// TIA Portal project "s7_1200_1214DCDCDC_loadcell_advanced" (V17)

(* hardware
DEVICE "S7-1200 station_1"  S7-1200 Station
   slot 0: "Rack_0"  S7-1200 Rack  Rack  V1.0
   slot 1: "PLC_1"  CPU 1214C DC/DC/DC  6ES7 214-1AG40-0XB0  V4.2
*)

// ===== PLC "PLC_1"  CPU 1214C DC/DC/DC =====

VAR_GLOBAL   // PLC tag table "Default tag table"
   "Start" AT %I0.2 : Bool;
   "Stop" AT %I0.3 : Bool;
   "Sensor_loadcell_in" AT %IW64 : UInt;
   "Sensor_Loadcell" AT %I0.4 : Bool;
   "Sensor_Classification" AT %I0.5 : Bool;
   "Cylinder_Push" AT %Q0.1 : Bool;
   "Cylinder_GoBack" AT %Q0.2 : Bool;
   "VEL" AT %MW160 : Int;
   "Tag_1" AT %M0.0 : Bool;
   "Tag_2" AT %M0.1 : Bool;
   "Tag_3" AT %M0.2 : Bool;
   "Tag_4" AT %M0.3 : Bool;
   "Tag_5" AT %M0.4 : Bool;
   "Sensor_Mass_Dectect" AT %I0.6 : Bool;
   "Tag_6" AT %M0.5 : Bool;
   "Tag_7" AT %M0.6 : Bool;
   "Tag_8" AT %MD20 : Real;
   "Tag_9" AT %MD30 : Real;
   "Tag_10" AT %MD40 : Real;
   "Tag_11" AT %MD50 : DInt;
   "Mass" AT %MW10 : Word;
   "System_Byte" AT %MB1 : Byte;
   "FirstScan" AT %M1.0 : Bool;
   "DiagStatusUpdate" AT %M1.1 : Bool;
   "AlwaysTRUE" AT %M1.2 : Bool;
   "AlwaysFALSE" AT %M1.3 : Bool;
   "Clock_Byte" AT %MB2 : Byte;
   "Clock_10Hz" AT %M2.0 : Bool;
   "Clock_5Hz" AT %M2.1 : Bool;
   "Clock_2.5Hz" AT %M2.2 : Bool;
   "Clock_2Hz" AT %M2.3 : Bool;
   "Clock_1.25Hz" AT %M2.4 : Bool;
   "Clock_1Hz" AT %M2.5 : Bool;
   "Clock_0.625Hz" AT %M2.6 : Bool;
   "Clock_0.5Hz" AT %M2.7 : Bool;
   "Tag_12" AT %MW12 : UInt;
   "Tag_13" AT %MW14 : UInt;
   "Counter" AT %MB10 : USInt;
   "Aver_val" AT %MW16 : UInt;
   "Tag_14" AT %MD44 : Real;
   "Tag_29" AT %MD48 : Real;
   "Tag_15" AT %M0.7 : Bool;
   "Tag_16" AT %MW18 : Word;
   "CV" AT %MD52 : Real;
   "Tag_20" AT %MD56 : Real;
   "RL_chan" AT %M3.1 : Bool;
   "RL_le" AT %M3.2 : Bool;
   "Tag_23" AT %M3.3 : Bool;
   "Tag_24" AT %M3.4 : Bool;
   "Tag_25" AT %MD60 : Real;
   "Tag_26" AT %MD64 : Real;
   "Mass_out_1" AT %MD66 : Real;
   "Mass_out_2" AT %MD70 : Real;
   "Tag_18" AT %M3.5 : Bool;
   "Tag_17" AT %M3.6 : Bool;
   "Tag_19" AT %M3.7 : Bool;
   "Tag_27" AT %M4.1 : Bool;
   "Tag_21" AT %Q0.3 : Bool;
   "Tag_22" AT %MD57 : Real;
   "Tag_28" AT %MD58 : Real;
   "Tag_30" AT %MD100 : Real;
   "Tag_31" AT %MD101 : Real;
   "Tag_32" AT %MD102 : Real;
   "Tag_33" AT %MD104 : Real;
   "Tag_34" AT %MD108 : Real;
   "Tag_35" AT %MD112 : Real;
   "Tag_36" AT %MD120 : DWord;
   "Tag_37" AT %MD124 : DWord;
   "Tag_38" AT %M4.2 : Bool;
   "Tag_39" AT %M4.4 : Bool;
   "Tag_40" AT %M4.3 : Bool;
END_VAR

DATA_BLOCK "Data_block_1"   // DB1
{ S7_Optimized_Access := 'FALSE' }
VERSION : 0.1
   VAR
      Pulse : Bool;
   END_VAR
BEGIN
END_DATA_BLOCK

// folder: System blocks/Program resources

DATA_BLOCK "CTU_02"   // DB2
{ S7_Optimized_Access := 'TRUE' }
AUTHOR : Simatic
FAMILY : IEC
NAME : CNTR
VERSION : 1.0
// stored: InstanceOfName IEC_COUNTER
"IEC_COUNTER"
BEGIN
END_DATA_BLOCK

DATA_BLOCK "CTU1"   // DB3
{ S7_Optimized_Access := 'TRUE' }
AUTHOR : Simatic
FAMILY : IEC
NAME : UDCNTR
VERSION : 1.2
// stored: InstanceOfName IEC_UDCOUNTER
"IEC_UDCOUNTER"
BEGIN
END_DATA_BLOCK

DATA_BLOCK "Timer_0"   // DB4
{ S7_Optimized_Access := 'TRUE' }
AUTHOR : Simatic
FAMILY : IEC
NAME : IEC_TMR
VERSION : 1.0
// stored: InstanceOfName IEC_TIMER
"IEC_TIMER"
BEGIN
END_DATA_BLOCK

DATA_BLOCK "Timer_1"   // DB5
{ S7_Optimized_Access := 'TRUE' }
AUTHOR : Simatic
FAMILY : IEC
NAME : IEC_TMR
VERSION : 1.0
// stored: InstanceOfName IEC_TIMER
"IEC_TIMER"
BEGIN
END_DATA_BLOCK

DATA_BLOCK "CTU_03"   // DB6
{ S7_Optimized_Access := 'TRUE' }
AUTHOR : Simatic
FAMILY : IEC
NAME : CNTR
VERSION : 1.0
// stored: InstanceOfName IEC_COUNTER
"IEC_COUNTER"
BEGIN
END_DATA_BLOCK

// folder: (top level)

FUNCTION "Block_1" : Void   // FC1, SCL
{ S7_Optimized_Access := 'TRUE' }
VERSION : 0.1
BEGIN
END_FUNCTION

ORGANIZATION_BLOCK "Main"   // OB1, LAD, ProgramCycle
TITLE = "Main Program Sweep (Cycle)"
{ S7_Optimized_Access := 'TRUE' }
VERSION : 0.1
   VAR_INPUT
      Initial_Call : Bool;   // Initial call of this OB
      Remanence : Bool;   // =True, if remanent data are available
   END_VAR
   VAR_TEMP   // added for the SCL form of the ladder/FBD networks
      _w1 : Bool;
      _w2 : Bool;
   END_VAR
BEGIN

REGION Network 1
   // POWER_ON/OFF
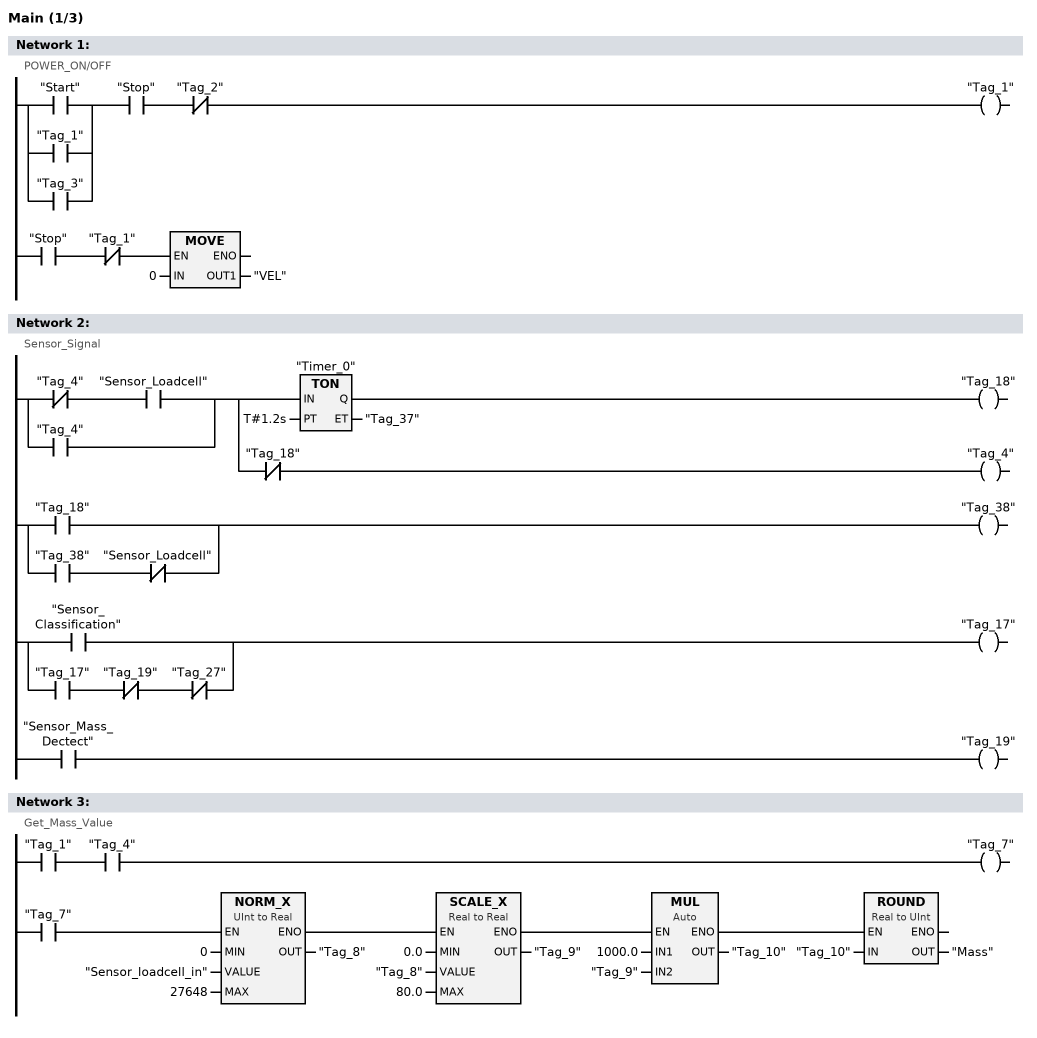
   RUNG wire#powerrail
      Contact( "Start" )
      wire#w1
      Contact( "Stop" )
      I_Contact( "Tag_2" )
      Coil( "Tag_1" )
   END_RUNG
   RUNG wire#powerrail
      Contact( "Tag_1" )
   END_RUNG wire#w1
   RUNG wire#powerrail
      Contact( "Tag_3" )
   END_RUNG wire#w1
   RUNG wire#powerrail
      Contact( "Stop" )
      I_Contact( "Tag_1" )
      Move(in := 0, out1 => "VEL")
   END_RUNG
   // the same network as SCL:
   "Tag_1" := ("Start" OR "Tag_1" OR "Tag_3") AND "Stop" AND NOT "Tag_2";
   IF "Stop" AND NOT "Tag_1" THEN "VEL" := 0; END_IF;
END_REGION

REGION Network 2
   // Sensor_Signal
   #_w1 := (NOT "Tag_4" AND "Sensor_Loadcell") OR "Tag_4";
   "Timer_0".TON(IN := #_w1, PT := T#1.2s, ET => "Tag_37");
   "Tag_18" := "Timer_0".Q;
   "Tag_4" := #_w1 AND NOT "Tag_18";
   "Tag_38" := "Tag_18" OR ("Tag_38" AND NOT "Sensor_Loadcell");
   "Tag_17" := "Sensor_Classification" OR ("Tag_17" AND NOT "Tag_19" AND NOT "Tag_27");
   "Tag_19" := "Sensor_Mass_Dectect";
END_REGION

REGION Network 3
   // Get_Mass_Value
   RUNG wire#powerrail
      Contact( "Tag_1" )
      Contact( "Tag_4" )
      Coil( "Tag_7" )
   END_RUNG
   RUNG wire#powerrail
      Contact( "Tag_7" )
      { S7_Templates := "[SrcType := UInt, DestType := Real]" } Normalize(min := 0, value := "Sensor_loadcell_in", max := 27648, out => "Tag_8")
      { S7_Templates := "[SrcType := Real, DestType := Real]" } Scale(min := 0.0, value := "Tag_8", max := 80.0, out => "Tag_9")
      Mul(in1 := 1000.0, in2 := "Tag_9", out => "Tag_10")
      { S7_Templates := "[SrcType := Real, DestType := UInt]" } Round(in := "Tag_10", out => "Mass")
   END_RUNG
   // the same network as SCL:
   "Tag_7" := "Tag_1" AND "Tag_4";
   IF "Tag_7" THEN
       "Tag_8" := NORM_X(MIN := 0, VALUE := "Sensor_loadcell_in", MAX := 27648);
       "Tag_9" := SCALE_X(MIN := 0.0, VALUE := "Tag_8", MAX := 80.0);
       "Tag_10" := 1000.0 * "Tag_9";
       "Mass" := ROUND("Tag_10");
   END_IF;
END_REGION

REGION Network 4
   // CALCULATE_AVER_MASS
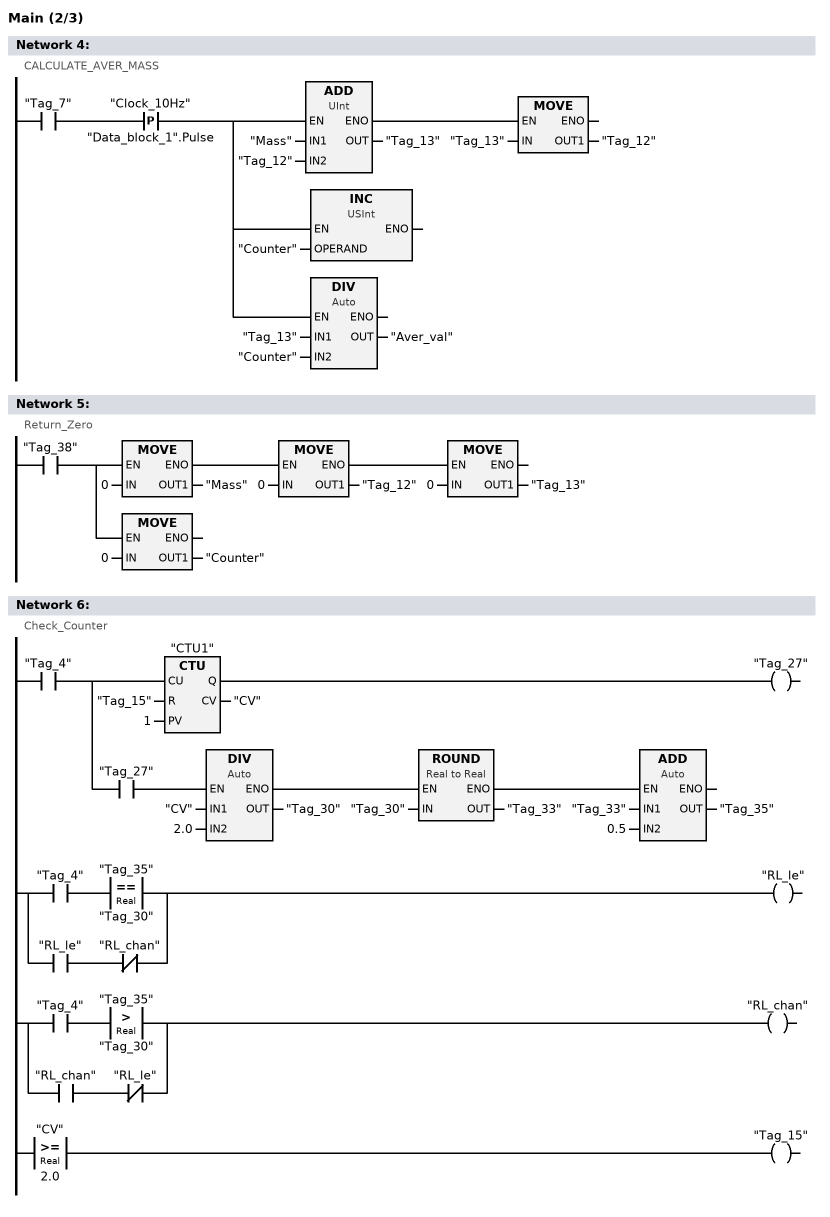
   RUNG wire#powerrail
      Contact( "Tag_7" )
      P_Contact(operand := "Clock_10Hz", bit := "Data_block_1".Pulse)
      wire#w1
      { S7_Templates := "SrcType := UInt" } Add(in1 := "Mass", in2 := "Tag_12", out => "Tag_13")
      Move(in := "Tag_13", out1 => "Tag_12")
   END_RUNG
   RUNG wire#w1
      { S7_Templates := "DestType := USInt" } Inc( "Counter" )
   END_RUNG
   RUNG wire#w1
      Div(in1 := "Tag_13", in2 := "Counter", out => "Aver_val")
   END_RUNG
   // the same network as SCL:
   #_w1 := "Tag_7" AND "Clock_10Hz" AND NOT "Data_block_1".Pulse;   // rising edge of "Clock_10Hz"
   "Data_block_1".Pulse := "Clock_10Hz";
   IF #_w1 THEN
       "Tag_13" := "Mass" + "Tag_12";
       "Tag_12" := "Tag_13";
       "Counter" := "Counter" + 1;
       "Aver_val" := "Tag_13" / "Counter";
   END_IF;
END_REGION

REGION Network 5
   // Return_Zero
   RUNG wire#powerrail
      Contact( "Tag_38" )
      wire#w1
      Move(in := 0, out1 => "Mass")
      Move(in := 0, out1 => "Tag_12")
      Move(in := 0, out1 => "Tag_13")
   END_RUNG
   RUNG wire#w1
      Move(in := 0, out1 => "Counter")
   END_RUNG
   // the same network as SCL:
   IF "Tag_38" THEN
       "Mass" := 0;
       "Tag_12" := 0;
       "Tag_13" := 0;
       "Counter" := 0;
   END_IF;
END_REGION

REGION Network 6
   // Check_Counter
   "CTU1".CTU(CU := "Tag_4", R := "Tag_15", PV := 1, CV => "CV");
   "Tag_27" := "CTU1".Q;
   IF "Tag_4" AND "Tag_27" THEN
       "Tag_30" := "CV" / 2.0;
       "Tag_33" := ROUND("Tag_30");
       "Tag_35" := "Tag_33" + 0.5;
   END_IF;
   "RL_le" := ("Tag_4" AND ("Tag_35" = "Tag_30")) OR ("RL_le" AND NOT "RL_chan");
   "RL_chan" := ("Tag_4" AND ("Tag_35" > "Tag_30")) OR ("RL_chan" AND NOT "RL_le");
   "Tag_15" := "CV" >= 2.0;
END_REGION

REGION Network 8
   // Function_Application
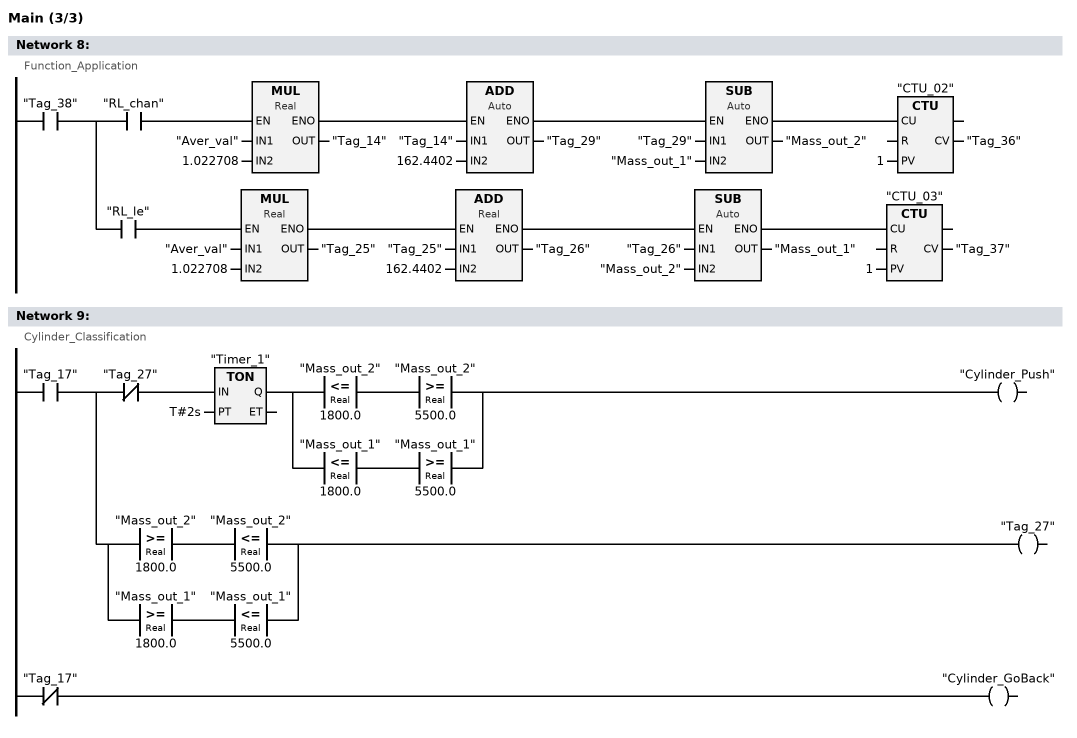
   #_w1 := "Tag_38" AND "RL_chan";
   IF #_w1 THEN
       "Tag_14" := "Aver_val" * 1.022708;
       "Tag_29" := "Tag_14" + 162.4402;
       "Mass_out_2" := "Tag_29" - "Mass_out_1";
   END_IF;
   "CTU_02".CTU(CU := #_w1, PV := 1, CV => "Tag_36");
   #_w2 := "Tag_38" AND "RL_le";
   IF #_w2 THEN
       "Tag_25" := "Aver_val" * 1.022708;
       "Tag_26" := "Tag_25" + 162.4402;
       "Mass_out_1" := "Tag_26" - "Mass_out_2";
   END_IF;
   "CTU_03".CTU(CU := #_w2, PV := 1, CV => "Tag_37");
END_REGION

REGION Network 9
   // Cylinder_Classification
   "Timer_1".TON(IN := "Tag_17" AND NOT "Tag_27", PT := T#2s);
   "Cylinder_Push" := "Timer_1".Q AND ((("Mass_out_2" <= 1800.0) AND ("Mass_out_2" >= 5500.0)) OR (("Mass_out_1" <= 1800.0) AND ("Mass_out_1" >= 5500.0)));
   "Tag_27" := "Tag_17" AND ((("Mass_out_2" >= 1800.0) AND ("Mass_out_2" <= 5500.0)) OR (("Mass_out_1" >= 1800.0) AND ("Mass_out_1" <= 5500.0)));
   "Cylinder_GoBack" := NOT "Tag_17";
END_REGION
END_ORGANIZATION_BLOCK